{attribute 'pack_mode':='1'}
TYPE OutboundToteParams :
STRUCT
	source_id : ModelIdentifier; // Identifier for the source inbound line.
	target_id : ModelIdentifier; // Identifier for the target work position.
END_STRUCT
END_TYPE

(* stored: Version 1.1.0.1, ProductVersion 3.1.4024.12
   DUT OutboundToteParams: Id {31e82e3b-b811-47f0-ac12-f89be84462fd} *)
